FUNCTION_BLOCK FB_MUL_UINT (* UINTMultiplication *)
  (* Standard: 61499-1-D.1; Classification: Math *)
  (* Version 0.1, 2001-08-03, JHC, Rockwell Automation, Simplified version *)
  (* Version 0.0, 1998-04-15, JHC, Rockwell Automation, Original version *)
  (* Compiler header: package fb.rt.vmath; *)
  (* Compiler Java IBM VisualAge 3.0 *)
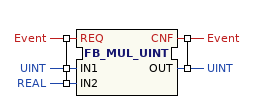
  EVENT_INPUT
    REQ WITH IN1, IN2;
  END_EVENT
  EVENT_OUTPUT
    CNF WITH OUT;
  END_EVENT
  VAR_INPUT
    IN1 : UINT; (* Augend *)
    IN2 : REAL; (* Addend *)
  END_VAR
  VAR_OUTPUT
    OUT : UINT; (* Sum *)
  END_VAR
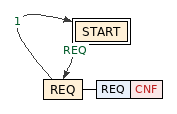
  EC_STATES
    START; (* Initial State *)
    REQ : REQ -> CNF; (* Normal execution *)
  END_STATES
  EC_TRANSITIONS
    START TO REQ := REQ;
    REQ TO START := 1;
  END_TRANSITIONS
  ALGORITHM REQ IN Java: (* Normally executed algorithm *)
OUT.value=(int)(IN1.value*IN2.value);
  END_ALGORITHM
END_FUNCTION_BLOCK
